FUNCTION F_StartsWith : BOOL
VAR_INPUT
    s      : STRING;
    prefix : STRING;
END_VAR

END_FUNCTION

(* stored: Version 1.1.0.1
   POU F_StartsWith: Id {96153f37-1b5d-43e0-bc68-5b729921d176}, SpecialFunc None *)
